FUNCTION TryConvert_SINT_TO_DATE : BOOL
VAR_INPUT
	in : SINT;
	out : REFERENCE TO DATE;
END_VAR

IF in < DatatypeLimits.MIN_VALUE_OF_SINT_WHICH_CAN_BE_HELD_IN_A_DATE THEN
	RETURN;
END_IF

out := SINT_TO_DATE(in);
TryConvert_SINT_TO_DATE := TRUE;

END_FUNCTION

(* stored: Version 1.1.0.1, ProductVersion 3.1.4024.12
   POU TryConvert_SINT_TO_DATE: Id {26d8514d-88a6-4d7b-a954-505b4a891890}, SpecialFunc None *)
